(* CODESYS project testLD_RECOVERED_2018-03-27T13-50-33.project

Project tree, tasks and I/O mapping:
  Device : Jinan Cherry-ARM Cortex-VxWorks, Jinan Cheery Electric Co., Ltd., version 3.5.11.20
    application Application
      libraries: Standard, * (System)
      task MainTask (cyclic, interval 4 ms, priority 1) calls PLC_PRG
      task EtherCAT_Task (cyclic, interval t#4ms, priority 1) calls nothing
      program PLC_PRG [FBD]
    SoftMotion General Axis Pool
    EtherCAT_Master : EtherCAT Master, 3S - Smart Software Solutions GmbH, version 3.5.12.0
        settings: NetworkName = 'gem1'; NetworkName = "gem1"; SrcAddress1 = 10; SrcAddress2 = 889192739
      FR8200 : EtherCAT Adapter, Huatai-smartLink, order no. FR8200, version Revision=16#00010001
          settings: ModularDevice = True; Number of Outputs = 0; Number of Inputs = 0; Number of Infos about Outputs = 0; Number of Infos about Inputs = 0; MDP_InputOffsets = [0,0,32,64,80]; MDP_OutputOffsets = [0,0,0,0,16]; StationAlias = 0; Sync.Length = 4; Sync.Length = 12; FMMU.Length = 4; FMMU.Length = 12; Number of RxPDOs of the Slave = 2; Number of TxPDOs of the Slave = 4; DC sync0 cycletime = 4000; DC sync1 cycletime = 4000; Number of SDO = 4; Command_0.Index = 16#8000; Command_0.Subindex = 16#01; Command_0.Value = 6; Command_0.Size = 16; Command_0.AbortIfError = FALSE; Command_0.JumpToLine = FALSE; Command_0.Line = 0; Command_0.CompleteAccess = False; Command_0.Index = 16#8010; Command_0.Subindex = 16#01; Command_0.Value = 6; Command_0.Size = 16; Command_0.AbortIfError = FALSE; Command_0.JumpToLine = FALSE; Command_0.Line = 0; Command_0.CompleteAccess = False; Command_0.Index = 16#8020; Command_0.Subindex = 16#01; Command_0.Value = 12; Command_0.Size = 16; Command_0.AbortIfError = FALSE; Command_0.JumpToLine = FALSE; Command_0.Line = 0;
            Command_0.CompleteAccess = False; Command_0.Index = 16#8030; Command_0.Subindex = 16#01; Command_0.Value = 12; Command_0.Size = 16; Command_0.AbortIfError = FALSE; Command_0.JumpToLine = FALSE; Command_0.Line = 0; Command_0.CompleteAccess = False; RxTxPdo.NumberofExcludes = 0; RxTxPdo.NumberofEntries = 9; RxTxPdo.Index = 16#1602; RxTxPdo.Fixed = False; RxTxPdo.Mandatory = False; RxTxPdo.Virtual = False; RxTxPdo.Sm = 2; RxTxPdo.Su = 0; RxTxPdo.Name = 'Channels Data'; RxTxPdo.DependOnSlot = True; RxTxPdo.DependOnSlotGroup = False; RxTxPdo.OverwrittenByModule = True; Channel 1.Index = 16#7040; Channel 1.SubIndex = 1; Channel 1.Size = 1; Channel 1.Offset = 0; Channel 1.DependOnSlot = True; Channel 1.DependOnSlotGroup = True; Channel 2.Index = 16#7040; Channel 2.SubIndex = 2; Channel 2.Size = 1; Channel 2.Offset = 0; Channel 2.DependOnSlot = True; Channel 2.DependOnSlotGroup = True; Channel 3.Index = 16#7040; Channel 3.SubIndex = 3; Channel 3.Size = 1; Channel 3.Offset = 0; Channel 3.DependOnSlot = True; Channel 3.DependOnSlotGroup = True; Channel 4.Index = 16#7040;
            Channel 4.SubIndex = 4; Channel 4.Size = 1; Channel 4.Offset = 0; Channel 4.DependOnSlot = True; Channel 4.DependOnSlotGroup = True; Channel 5.Index = 16#7040; Channel 5.SubIndex = 5; Channel 5.Size = 1; Channel 5.Offset = 0; Channel 5.DependOnSlot = True; Channel 5.DependOnSlotGroup = True; Channel 6.Index = 16#7040; Channel 6.SubIndex = 6; Channel 6.Size = 1; Channel 6.Offset = 0; Channel 6.DependOnSlot = True; Channel 6.DependOnSlotGroup = True; Channel 7.Index = 16#7040; Channel 7.SubIndex = 7; Channel 7.Size = 1; Channel 7.Offset = 0; Channel 7.DependOnSlot = True; Channel 7.DependOnSlotGroup = True; Channel 8.Index = 16#7040; Channel 8.SubIndex = 8; Channel 8.Size = 1; Channel 8.Offset = 0; Channel 8.DependOnSlot = True; Channel 8.DependOnSlotGroup = True; Entry.Index = 16#0000; Entry.SubIndex = 9; Entry.Size = 8; Entry.Offset = 0; Entry.DependOnSlot = True; Entry.DependOnSlotGroup = True; RxTxPdo.NumberofExcludes = 0; RxTxPdo.NumberofEntries = 9; RxTxPdo.Index = 16#1603; RxTxPdo.Fixed = False; RxTxPdo.Mandatory = False;
            RxTxPdo.Virtual = False; RxTxPdo.Sm = 2; RxTxPdo.Su = 0; RxTxPdo.Name = 'Channels Data'; RxTxPdo.DependOnSlot = True; RxTxPdo.DependOnSlotGroup = False; RxTxPdo.OverwrittenByModule = True; Channel 1.Index = 16#7030; Channel 1.SubIndex = 1; Channel 1.Size = 1; Channel 1.Offset = 0; Channel 1.DependOnSlot = True; Channel 1.DependOnSlotGroup = True; Channel 2.Index = 16#7030; Channel 2.SubIndex = 2; Channel 2.Size = 1; Channel 2.Offset = 0; Channel 2.DependOnSlot = True; Channel 2.DependOnSlotGroup = True; Channel 3.Index = 16#7030; Channel 3.SubIndex = 3; Channel 3.Size = 1; Channel 3.Offset = 0; Channel 3.DependOnSlot = True; Channel 3.DependOnSlotGroup = True; Channel 4.Index = 16#7030; Channel 4.SubIndex = 4; Channel 4.Size = 1; Channel 4.Offset = 0; Channel 4.DependOnSlot = True; Channel 4.DependOnSlotGroup = True; Channel 5.Index = 16#7030; Channel 5.SubIndex = 5; Channel 5.Size = 1; Channel 5.Offset = 0; Channel 5.DependOnSlot = True; Channel 5.DependOnSlotGroup = True; Channel 6.Index = 16#7030; Channel 6.SubIndex = 6; Channel 6.Size = 1;
            Channel 6.Offset = 0; Channel 6.DependOnSlot = True; Channel 6.DependOnSlotGroup = True; Channel 7.Index = 16#7030; Channel 7.SubIndex = 7; Channel 7.Size = 1; Channel 7.Offset = 0; Channel 7.DependOnSlot = True; Channel 7.DependOnSlotGroup = True; Channel 8.Index = 16#7030; Channel 8.SubIndex = 8; Channel 8.Size = 1; Channel 8.Offset = 0; Channel 8.DependOnSlot = True; Channel 8.DependOnSlotGroup = True; Entry.Index = 16#0000; Entry.SubIndex = 9; Entry.Size = 8; Entry.Offset = 0; Entry.DependOnSlot = True; Entry.DependOnSlotGroup = True; RxTxPdo.NumberofExcludes = 0; RxTxPdo.NumberofEntries = 12; RxTxPdo.Index = 16#1A00; RxTxPdo.Fixed = False; RxTxPdo.Mandatory = False; RxTxPdo.Virtual = False; RxTxPdo.Sm = 3; RxTxPdo.Su = 0; RxTxPdo.Name = 'Channels Data'; RxTxPdo.DependOnSlot = True; RxTxPdo.DependOnSlotGroup = False; RxTxPdo.OverwrittenByModule = True; Channel 1.Index = 16#6000; Channel 1.SubIndex = 1; Channel 1.Size = 1; Channel 1.Offset = 0; Channel 1.DependOnSlot = True; Channel 1.DependOnSlotGroup = True; Channel 2.Index = 16#6000;
            Channel 2.SubIndex = 2; Channel 2.Size = 1; Channel 2.Offset = 0; Channel 2.DependOnSlot = True; Channel 2.DependOnSlotGroup = True; Channel 3.Index = 16#6000; Channel 3.SubIndex = 3; Channel 3.Size = 1; Channel 3.Offset = 0; Channel 3.DependOnSlot = True; Channel 3.DependOnSlotGroup = True; Channel 4.Index = 16#6000; Channel 4.SubIndex = 4; Channel 4.Size = 1; Channel 4.Offset = 0; Channel 4.DependOnSlot = True; Channel 4.DependOnSlotGroup = True; Channel 5.Index = 16#6000; Channel 5.SubIndex = 5; Channel 5.Size = 1; Channel 5.Offset = 0; Channel 5.DependOnSlot = True; Channel 5.DependOnSlotGroup = True; Channel 6.Index = 16#6000; Channel 6.SubIndex = 6; Channel 6.Size = 1; Channel 6.Offset = 0; Channel 6.DependOnSlot = True; Channel 6.DependOnSlotGroup = True; Channel 7.Index = 16#6000; Channel 7.SubIndex = 7; Channel 7.Size = 1; Channel 7.Offset = 0; Channel 7.DependOnSlot = True; Channel 7.DependOnSlotGroup = True; Channel 8.Index = 16#6000; Channel 8.SubIndex = 8; Channel 8.Size = 1; Channel 8.Offset = 0; Channel 8.DependOnSlot = True;
            Channel 8.DependOnSlotGroup = True; Entry.Index = 16#0000; Entry.SubIndex = 9; Entry.Size = 8; Entry.Offset = 0; Entry.DependOnSlot = True; Entry.DependOnSlotGroup = True; Temperature Alarm.Index = 16#6002; Temperature Alarm.SubIndex = 1; Temperature Alarm.Size = 1; Temperature Alarm.Offset = 0; Temperature Alarm.DependOnSlot = True; Temperature Alarm.DependOnSlotGroup = True; Voltage Alarm.Index = 16#6002; Voltage Alarm.SubIndex = 2; Voltage Alarm.Size = 1; Voltage Alarm.Offset = 0; Voltage Alarm.DependOnSlot = True; Voltage Alarm.DependOnSlotGroup = True; Entry.Index = 16#0000; Entry.SubIndex = 3; Entry.Size = 14; Entry.Offset = 0; Entry.DependOnSlot = False; Entry.DependOnSlotGroup = False; RxTxPdo.NumberofExcludes = 0; RxTxPdo.NumberofEntries = 12; RxTxPdo.Index = 16#1A01; RxTxPdo.Fixed = False; RxTxPdo.Mandatory = False; RxTxPdo.Virtual = False; RxTxPdo.Sm = 3; RxTxPdo.Su = 0; RxTxPdo.Name = 'Channels Data'; RxTxPdo.DependOnSlot = True; RxTxPdo.DependOnSlotGroup = False; RxTxPdo.OverwrittenByModule = True; Channel 1.Index = 16#6010; Channel 1.SubIndex = 1; Channel 1.Size = 1;
            Channel 1.Offset = 0; Channel 1.DependOnSlot = True; Channel 1.DependOnSlotGroup = True; Channel 2.Index = 16#6010; Channel 2.SubIndex = 2; Channel 2.Size = 1; Channel 2.Offset = 0; Channel 2.DependOnSlot = True; Channel 2.DependOnSlotGroup = True; Channel 3.Index = 16#6010; Channel 3.SubIndex = 3; Channel 3.Size = 1; Channel 3.Offset = 0; Channel 3.DependOnSlot = True; Channel 3.DependOnSlotGroup = True; Channel 4.Index = 16#6010; Channel 4.SubIndex = 4; Channel 4.Size = 1; Channel 4.Offset = 0; Channel 4.DependOnSlot = True; Channel 4.DependOnSlotGroup = True; Channel 5.Index = 16#6010; Channel 5.SubIndex = 5; Channel 5.Size = 1; Channel 5.Offset = 0; Channel 5.DependOnSlot = True; Channel 5.DependOnSlotGroup = True; Channel 6.Index = 16#6010; Channel 6.SubIndex = 6; Channel 6.Size = 1; Channel 6.Offset = 0; Channel 6.DependOnSlot = True; Channel 6.DependOnSlotGroup = True; Channel 7.Index = 16#6010; Channel 7.SubIndex = 7; Channel 7.Size = 1; Channel 7.Offset = 0; Channel 7.DependOnSlot = True; Channel 7.DependOnSlotGroup = True; Channel 8.Index = 16#6010;
            Channel 8.SubIndex = 8; Channel 8.Size = 1; Channel 8.Offset = 0; Channel 8.DependOnSlot = True; Channel 8.DependOnSlotGroup = True; Entry.Index = 16#0000; Entry.SubIndex = 9; Entry.Size = 8; Entry.Offset = 0; Entry.DependOnSlot = True; Entry.DependOnSlotGroup = True; Temperature Alarm.Index = 16#6012; Temperature Alarm.SubIndex = 1; Temperature Alarm.Size = 1; Temperature Alarm.Offset = 0; Temperature Alarm.DependOnSlot = True; Temperature Alarm.DependOnSlotGroup = True; Voltage Alarm.Index = 16#6012; Voltage Alarm.SubIndex = 2; Voltage Alarm.Size = 1; Voltage Alarm.Offset = 0; Voltage Alarm.DependOnSlot = True; Voltage Alarm.DependOnSlotGroup = True; Entry.Index = 16#0000; Entry.SubIndex = 3; Entry.Size = 14; Entry.Offset = 0; Entry.DependOnSlot = False; Entry.DependOnSlotGroup = False; RxTxPdo.NumberofExcludes = 0; RxTxPdo.NumberofEntries = 3; RxTxPdo.Index = 16#1A02; RxTxPdo.Fixed = False; RxTxPdo.Mandatory = False; RxTxPdo.Virtual = False; RxTxPdo.Sm = 3; RxTxPdo.Su = 0; RxTxPdo.Name = 'Alarm Data'; RxTxPdo.DependOnSlot = True; RxTxPdo.DependOnSlotGroup = False;
            RxTxPdo.OverwrittenByModule = True; Temperature Alarm.Index = 16#6022; Temperature Alarm.SubIndex = 1; Temperature Alarm.Size = 1; Temperature Alarm.Offset = 0; Temperature Alarm.DependOnSlot = True; Temperature Alarm.DependOnSlotGroup = True; Voltage Alarm.Index = 16#6022; Voltage Alarm.SubIndex = 2; Voltage Alarm.Size = 1; Voltage Alarm.Offset = 0; Voltage Alarm.DependOnSlot = True; Voltage Alarm.DependOnSlotGroup = True; Entry.Index = 16#0000; Entry.SubIndex = 3; Entry.Size = 14; Entry.Offset = 0; Entry.DependOnSlot = False; Entry.DependOnSlotGroup = False; RxTxPdo.NumberofExcludes = 0; RxTxPdo.NumberofEntries = 3; RxTxPdo.Index = 16#1A03; RxTxPdo.Fixed = False; RxTxPdo.Mandatory = False; RxTxPdo.Virtual = False; RxTxPdo.Sm = 3; RxTxPdo.Su = 0; RxTxPdo.Name = 'Alarm Data'; RxTxPdo.DependOnSlot = True; RxTxPdo.DependOnSlotGroup = False; RxTxPdo.OverwrittenByModule = True; Temperature Alarm.Index = 16#6032; Temperature Alarm.SubIndex = 1; Temperature Alarm.Size = 1; Temperature Alarm.Offset = 0; Temperature Alarm.DependOnSlot = True; Temperature Alarm.DependOnSlotGroup = True; Voltage Alarm.Index = 16#6032; Voltage Alarm.SubIndex = 2; Voltage Alarm.Size = 1;
            Voltage Alarm.Offset = 0; Voltage Alarm.DependOnSlot = True; Voltage Alarm.DependOnSlotGroup = True; Entry.Index = 16#0000; Entry.SubIndex = 3; Entry.Size = 14; Entry.Offset = 0; Entry.DependOnSlot = False; Entry.DependOnSlotGroup = False; Channel 1.Name = 'Channel 1'; Channel 1.DataType = 'BOOL'; Channel 1.Default = ''; Channel 1.Comment = ''; Channel 2.Name = 'Channel 2'; Channel 2.DataType = 'BOOL'; Channel 2.Default = ''; Channel 2.Comment = ''; Channel 3.Name = 'Channel 3'; Channel 3.DataType = 'BOOL'; Channel 3.Default = ''; Channel 3.Comment = ''; Channel 4.Name = 'Channel 4'; Channel 4.DataType = 'BOOL'; Channel 4.Default = ''; Channel 4.Comment = ''; Channel 5.Name = 'Channel 5'; Channel 5.DataType = 'BOOL'; Channel 5.Default = ''; Channel 5.Comment = ''; Channel 6.Name = 'Channel 6'; Channel 6.DataType = 'BOOL'; Channel 6.Default = ''; Channel 6.Comment = ''; Channel 7.Name = 'Channel 7'; Channel 7.DataType = 'BOOL'; Channel 7.Default = ''; Channel 7.Comment = ''; Channel 8.Name = 'Channel 8'; Channel 8.DataType = 'BOOL'; Channel 8.Default = '';
            Channel 8.Comment = ''; Entry.Name = ''; Entry.DataType = ''; Entry.Default = ''; Entry.Comment = ''; Channel 1.Name = 'Channel 1'; Channel 1.DataType = 'BOOL'; Channel 1.Default = ''; Channel 1.Comment = ''; Channel 2.Name = 'Channel 2'; Channel 2.DataType = 'BOOL'; Channel 2.Default = ''; Channel 2.Comment = ''; Channel 3.Name = 'Channel 3'; Channel 3.DataType = 'BOOL'; Channel 3.Default = ''; Channel 3.Comment = ''; Channel 4.Name = 'Channel 4'; Channel 4.DataType = 'BOOL'; Channel 4.Default = ''; Channel 4.Comment = ''; Channel 5.Name = 'Channel 5'; Channel 5.DataType = 'BOOL'; Channel 5.Default = ''; Channel 5.Comment = ''; Channel 6.Name = 'Channel 6'; Channel 6.DataType = 'BOOL'; Channel 6.Default = ''; Channel 6.Comment = ''; Channel 7.Name = 'Channel 7'; Channel 7.DataType = 'BOOL'; Channel 7.Default = ''; Channel 7.Comment = ''; Channel 8.Name = 'Channel 8'; Channel 8.DataType = 'BOOL'; Channel 8.Default = ''; Channel 8.Comment = ''; Entry.Name = ''; Entry.DataType = ''; Entry.Default = '';
            Entry.Comment = ''; Channel 1.Name = 'Channel 1'; Channel 1.DataType = 'BOOL'; Channel 1.Default = ''; Channel 1.Comment = ''; Channel 2.Name = 'Channel 2'; Channel 2.DataType = 'BOOL'; Channel 2.Default = ''; Channel 2.Comment = ''; Channel 3.Name = 'Channel 3'; Channel 3.DataType = 'BOOL'; Channel 3.Default = ''; Channel 3.Comment = ''; Channel 4.Name = 'Channel 4'; Channel 4.DataType = 'BOOL'; Channel 4.Default = ''; Channel 4.Comment = ''; Channel 5.Name = 'Channel 5'; Channel 5.DataType = 'BOOL'; Channel 5.Default = ''; Channel 5.Comment = ''; Channel 6.Name = 'Channel 6'; Channel 6.DataType = 'BOOL'; Channel 6.Default = ''; Channel 6.Comment = ''; Channel 7.Name = 'Channel 7'; Channel 7.DataType = 'BOOL'; Channel 7.Default = ''; Channel 7.Comment = ''; Channel 8.Name = 'Channel 8'; Channel 8.DataType = 'BOOL'; Channel 8.Default = ''; Channel 8.Comment = ''; Entry.Name = ''; Entry.DataType = ''; Entry.Default = ''; Entry.Comment = ''; Temperature Alarm.Name = 'Temperature Alarm'; Temperature Alarm.DataType = 'BOOL'; Temperature Alarm.Default = '';
            Temperature Alarm.Comment = ''; Voltage Alarm.Name = 'Voltage Alarm'; Voltage Alarm.DataType = 'BOOL'; Voltage Alarm.Default = ''; Voltage Alarm.Comment = ''; Entry.Name = ''; Entry.DataType = ''; Entry.Default = ''; Entry.Comment = ''; Channel 1.Name = 'Channel 1'; Channel 1.DataType = 'BOOL'; Channel 1.Default = ''; Channel 1.Comment = ''; Channel 2.Name = 'Channel 2'; Channel 2.DataType = 'BOOL'; Channel 2.Default = ''; Channel 2.Comment = ''; Channel 3.Name = 'Channel 3'; Channel 3.DataType = 'BOOL'; Channel 3.Default = ''; Channel 3.Comment = ''; Channel 4.Name = 'Channel 4'; Channel 4.DataType = 'BOOL'; Channel 4.Default = ''; Channel 4.Comment = ''; Channel 5.Name = 'Channel 5'; Channel 5.DataType = 'BOOL'; Channel 5.Default = ''; Channel 5.Comment = ''; Channel 6.Name = 'Channel 6'; Channel 6.DataType = 'BOOL'; Channel 6.Default = ''; Channel 6.Comment = ''; Channel 7.Name = 'Channel 7'; Channel 7.DataType = 'BOOL'; Channel 7.Default = ''; Channel 7.Comment = ''; Channel 8.Name = 'Channel 8'; Channel 8.DataType = 'BOOL'; Channel 8.Default = '';
            Channel 8.Comment = ''; Entry.Name = ''; Entry.DataType = ''; Entry.Default = ''; Entry.Comment = ''; Temperature Alarm.Name = 'Temperature Alarm'; Temperature Alarm.DataType = 'BOOL'; Temperature Alarm.Default = ''; Temperature Alarm.Comment = ''; Voltage Alarm.Name = 'Voltage Alarm'; Voltage Alarm.DataType = 'BOOL'; Voltage Alarm.Default = ''; Voltage Alarm.Comment = ''; Entry.Name = ''; Entry.DataType = ''; Entry.Default = ''; Entry.Comment = ''; Temperature Alarm.Name = 'Temperature Alarm'; Temperature Alarm.DataType = 'BOOL'; Temperature Alarm.Default = ''; Temperature Alarm.Comment = ''; Voltage Alarm.Name = 'Voltage Alarm'; Voltage Alarm.DataType = 'BOOL'; Voltage Alarm.Default = ''; Voltage Alarm.Comment = ''; Entry.Name = ''; Entry.DataType = ''; Entry.Default = ''; Entry.Comment = ''; Temperature Alarm.Name = 'Temperature Alarm'; Temperature Alarm.DataType = 'BOOL'; Temperature Alarm.Default = ''; Temperature Alarm.Comment = ''; Voltage Alarm.Name = 'Voltage Alarm'; Voltage Alarm.DataType = 'BOOL'; Voltage Alarm.Default = ''; Voltage Alarm.Comment = ''; Entry.Name = ''; Entry.DataType = ''; Entry.Default = '';
            Entry.Comment = ''
        <空14>
        <空10>
        <空19>
        <空32>
        <空23>
        <空15>
        <空21>
        <空31>
        <空26>
        <空16>
        <空20>
        FR1118 : FR Serials IO Modules, Huatai-smartLink, order no. FR1118, version 0
            settings: Number of Inputs = 25; Number of Infos about Inputs = 25; Channel 1.Offset = 0; Channel 1.DependOnSlot = True; Channel 1.DependOnSlotGroup = True; Channel 2.Offset = 0; Channel 2.DependOnSlot = True; Channel 2.DependOnSlotGroup = True; Channel 3.Offset = 0; Channel 3.DependOnSlot = True; Channel 3.DependOnSlotGroup = True; Channel 4.Offset = 0; Channel 4.DependOnSlot = True; Channel 4.DependOnSlotGroup = True; Channel 5.Offset = 0; Channel 5.DependOnSlot = True; Channel 5.DependOnSlotGroup = True; Channel 6.Offset = 0; Channel 6.DependOnSlot = True; Channel 6.DependOnSlotGroup = True; Channel 7.Offset = 0; Channel 7.DependOnSlot = True; Channel 7.DependOnSlotGroup = True; Channel 8.Offset = 0; Channel 8.DependOnSlot = True; Channel 8.DependOnSlotGroup = True; Entry.Offset = 0; Entry.DependOnSlot = True; Entry.DependOnSlotGroup = True; Temperature Alarm.Offset = 0; Temperature Alarm.DependOnSlot = True; Temperature Alarm.DependOnSlotGroup = True; Voltage Alarm.Offset = 0; Voltage Alarm.DependOnSlot = True; Voltage Alarm.DependOnSlotGroup = True; Entry.Offset = 0; Entry.DependOnSlot = False; Entry.DependOnSlotGroup = False; Channel 1.Default = ''; Channel 2.Default = '';
              Channel 3.Default = ''; Channel 4.Default = ''; Channel 5.Default = ''; Channel 6.Default = ''; Channel 7.Default = ''; Channel 8.Default = ''; Entry.Name = ''; Entry.DataType = ''; Entry.Default = ''; Temperature Alarm.Default = ''; Voltage Alarm.Default = ''; Entry.Name = ''; Entry.DataType = ''; Entry.Default = ''
            unmapped channels: Channel 1, Channel 2, Channel 3, Channel 4, Channel 5, Channel 6, Channel 7, Channel 8, , Temperature Alarm, Voltage Alarm, , , , , , , , , , , , , , 
        <空29>
        FR1118_1 : FR Serials IO Modules, Huatai-smartLink, order no. FR1118, version 0
            settings: Number of Inputs = 25; Number of Infos about Inputs = 25; Channel 1.Index = 16#6010; Channel 1.SubIndex = 1; Channel 1.Size = 1; Channel 1.Offset = 0; Channel 1.DependOnSlot = True; Channel 1.DependOnSlotGroup = True; Channel 2.Index = 16#6010; Channel 2.SubIndex = 2; Channel 2.Size = 1; Channel 2.Offset = 0; Channel 2.DependOnSlot = True; Channel 2.DependOnSlotGroup = True; Channel 3.Index = 16#6010; Channel 3.SubIndex = 3; Channel 3.Size = 1; Channel 3.Offset = 0; Channel 3.DependOnSlot = True; Channel 3.DependOnSlotGroup = True; Channel 4.Index = 16#6010; Channel 4.SubIndex = 4; Channel 4.Size = 1; Channel 4.Offset = 0; Channel 4.DependOnSlot = True; Channel 4.DependOnSlotGroup = True; Channel 5.Index = 16#6010; Channel 5.SubIndex = 5; Channel 5.Size = 1; Channel 5.Offset = 0; Channel 5.DependOnSlot = True; Channel 5.DependOnSlotGroup = True; Channel 6.Index = 16#6010; Channel 6.SubIndex = 6; Channel 6.Size = 1; Channel 6.Offset = 0; Channel 6.DependOnSlot = True; Channel 6.DependOnSlotGroup = True; Channel 7.Index = 16#6010; Channel 7.SubIndex = 7;
              Channel 7.Size = 1; Channel 7.Offset = 0; Channel 7.DependOnSlot = True; Channel 7.DependOnSlotGroup = True; Channel 8.Index = 16#6010; Channel 8.SubIndex = 8; Channel 8.Size = 1; Channel 8.Offset = 0; Channel 8.DependOnSlot = True; Channel 8.DependOnSlotGroup = True; Entry.Index = 16#0000; Entry.SubIndex = 9; Entry.Size = 8; Entry.Offset = 0; Entry.DependOnSlot = True; Entry.DependOnSlotGroup = True; Temperature Alarm.Index = 16#6012; Temperature Alarm.SubIndex = 1; Temperature Alarm.Size = 1; Temperature Alarm.Offset = 0; Temperature Alarm.DependOnSlot = True; Temperature Alarm.DependOnSlotGroup = True; Voltage Alarm.Index = 16#6012; Voltage Alarm.SubIndex = 2; Voltage Alarm.Size = 1; Voltage Alarm.Offset = 0; Voltage Alarm.DependOnSlot = True; Voltage Alarm.DependOnSlotGroup = True; Entry.Index = 16#0000; Entry.SubIndex = 3; Entry.Size = 14; Entry.Offset = 0; Entry.DependOnSlot = False; Entry.DependOnSlotGroup = False; Channel 1.Name = 'Channel 1'; Channel 1.DataType = 'BOOL'; Channel 1.Default = ''; Channel 1.Comment = ''; Channel 2.Name = 'Channel 2'; Channel 2.DataType = 'BOOL';
              Channel 2.Default = ''; Channel 2.Comment = ''; Channel 3.Name = 'Channel 3'; Channel 3.DataType = 'BOOL'; Channel 3.Default = ''; Channel 3.Comment = ''; Channel 4.Name = 'Channel 4'; Channel 4.DataType = 'BOOL'; Channel 4.Default = ''; Channel 4.Comment = ''; Channel 5.Name = 'Channel 5'; Channel 5.DataType = 'BOOL'; Channel 5.Default = ''; Channel 5.Comment = ''; Channel 6.Name = 'Channel 6'; Channel 6.DataType = 'BOOL'; Channel 6.Default = ''; Channel 6.Comment = ''; Channel 7.Name = 'Channel 7'; Channel 7.DataType = 'BOOL'; Channel 7.Default = ''; Channel 7.Comment = ''; Channel 8.Name = 'Channel 8'; Channel 8.DataType = 'BOOL'; Channel 8.Default = ''; Channel 8.Comment = ''; Entry.Name = ''; Entry.DataType = ''; Entry.Default = ''; Entry.Comment = ''; Temperature Alarm.Name = 'Temperature Alarm'; Temperature Alarm.DataType = 'BOOL'; Temperature Alarm.Default = ''; Temperature Alarm.Comment = ''; Voltage Alarm.Name = 'Voltage Alarm'; Voltage Alarm.DataType = 'BOOL'; Voltage Alarm.Default = ''; Voltage Alarm.Comment = ''; Entry.Name = ''; Entry.DataType = '';
              Entry.Default = ''; Entry.Comment = ''
            unmapped channels: Channel 1, Channel 2, Channel 3, Channel 4, Channel 5, Channel 6, Channel 7, Channel 8, , Temperature Alarm, Voltage Alarm, , , , , , , , , , , , , , 
        <空18>
        <空22>
        <空7>
        <空5>
        <空11>
        FR2118_1 : FR Serials IO Modules, Huatai-smartLink, order no. FR2118, version 0
            settings: Number of Outputs = 9; Number of Inputs = 16; Number of Infos about Outputs = 9; Number of Infos about Inputs = 16; Channel 1.Index = 16#7030; Channel 1.SubIndex = 1; Channel 1.Size = 1; Channel 1.Offset = 0; Channel 1.DependOnSlot = True; Channel 1.DependOnSlotGroup = True; Channel 2.Index = 16#7030; Channel 2.SubIndex = 2; Channel 2.Size = 1; Channel 2.Offset = 0; Channel 2.DependOnSlot = True; Channel 2.DependOnSlotGroup = True; Channel 3.Index = 16#7030; Channel 3.SubIndex = 3; Channel 3.Size = 1; Channel 3.Offset = 0; Channel 3.DependOnSlot = True; Channel 3.DependOnSlotGroup = True; Channel 4.Index = 16#7030; Channel 4.SubIndex = 4; Channel 4.Size = 1; Channel 4.Offset = 0; Channel 4.DependOnSlot = True; Channel 4.DependOnSlotGroup = True; Channel 5.Index = 16#7030; Channel 5.SubIndex = 5; Channel 5.Size = 1; Channel 5.Offset = 0; Channel 5.DependOnSlot = True; Channel 5.DependOnSlotGroup = True; Channel 6.Index = 16#7030; Channel 6.SubIndex = 6; Channel 6.Size = 1; Channel 6.Offset = 0; Channel 6.DependOnSlot = True; Channel 6.DependOnSlotGroup = True;
              Channel 7.Index = 16#7030; Channel 7.SubIndex = 7; Channel 7.Size = 1; Channel 7.Offset = 0; Channel 7.DependOnSlot = True; Channel 7.DependOnSlotGroup = True; Channel 8.Index = 16#7030; Channel 8.SubIndex = 8; Channel 8.Size = 1; Channel 8.Offset = 0; Channel 8.DependOnSlot = True; Channel 8.DependOnSlotGroup = True; Entry.Index = 16#0000; Entry.SubIndex = 9; Entry.Size = 8; Entry.Offset = 0; Entry.DependOnSlot = True; Entry.DependOnSlotGroup = True; Temperature Alarm.Index = 16#6032; Temperature Alarm.SubIndex = 1; Temperature Alarm.Size = 1; Temperature Alarm.Offset = 0; Temperature Alarm.DependOnSlot = True; Temperature Alarm.DependOnSlotGroup = True; Voltage Alarm.Index = 16#6032; Voltage Alarm.SubIndex = 2; Voltage Alarm.Size = 1; Voltage Alarm.Offset = 0; Voltage Alarm.DependOnSlot = True; Voltage Alarm.DependOnSlotGroup = True; Entry.Index = 16#0000; Entry.SubIndex = 3; Entry.Size = 14; Entry.Offset = 0; Entry.DependOnSlot = False; Entry.DependOnSlotGroup = False; Channel 1.Name = 'Channel 1'; Channel 1.DataType = 'BOOL'; Channel 1.Default = ''; Channel 1.Comment = '';
              Channel 2.Name = 'Channel 2'; Channel 2.DataType = 'BOOL'; Channel 2.Default = ''; Channel 2.Comment = ''; Channel 3.Name = 'Channel 3'; Channel 3.DataType = 'BOOL'; Channel 3.Default = ''; Channel 3.Comment = ''; Channel 4.Name = 'Channel 4'; Channel 4.DataType = 'BOOL'; Channel 4.Default = ''; Channel 4.Comment = ''; Channel 5.Name = 'Channel 5'; Channel 5.DataType = 'BOOL'; Channel 5.Default = ''; Channel 5.Comment = ''; Channel 6.Name = 'Channel 6'; Channel 6.DataType = 'BOOL'; Channel 6.Default = ''; Channel 6.Comment = ''; Channel 7.Name = 'Channel 7'; Channel 7.DataType = 'BOOL'; Channel 7.Default = ''; Channel 7.Comment = ''; Channel 8.Name = 'Channel 8'; Channel 8.DataType = 'BOOL'; Channel 8.Default = ''; Channel 8.Comment = ''; Entry.Name = ''; Entry.DataType = ''; Entry.Default = ''; Entry.Comment = ''; Temperature Alarm.Name = 'Temperature Alarm'; Temperature Alarm.DataType = 'BOOL'; Temperature Alarm.Default = ''; Temperature Alarm.Comment = ''; Voltage Alarm.Name = 'Voltage Alarm'; Voltage Alarm.DataType = 'BOOL'; Voltage Alarm.Default = ''; Voltage Alarm.Comment = '';
              Entry.Name = ''; Entry.DataType = ''; Entry.Default = ''; Entry.Comment = ''
            output Application.PLC_PRG.Out1 : BIT  // Channel 1
            unmapped channels: Channel 2, Channel 3, Channel 4, Channel 5, Channel 6, Channel 7, Channel 8, , Temperature Alarm, Voltage Alarm, , , , , , , , , , , , , , 
        <空24>
        FR2118 : FR Serials IO Modules, Huatai-smartLink, order no. FR2118, version 0
            settings: Number of Outputs = 9; Number of Inputs = 16; Number of Infos about Outputs = 9; Number of Infos about Inputs = 16; Channel 1.Index = 16#7020; Channel 1.Offset = 0; Channel 1.DependOnSlot = True; Channel 1.DependOnSlotGroup = True; Channel 2.Index = 16#7020; Channel 2.Offset = 0; Channel 2.DependOnSlot = True; Channel 2.DependOnSlotGroup = True; Channel 3.Index = 16#7020; Channel 3.Offset = 0; Channel 3.DependOnSlot = True; Channel 3.DependOnSlotGroup = True; Channel 4.Index = 16#7020; Channel 4.Offset = 0; Channel 4.DependOnSlot = True; Channel 4.DependOnSlotGroup = True; Channel 5.Index = 16#7020; Channel 5.Offset = 0; Channel 5.DependOnSlot = True; Channel 5.DependOnSlotGroup = True; Channel 6.Index = 16#7020; Channel 6.Offset = 0; Channel 6.DependOnSlot = True; Channel 6.DependOnSlotGroup = True; Channel 7.Index = 16#7020; Channel 7.Offset = 0; Channel 7.DependOnSlot = True; Channel 7.DependOnSlotGroup = True; Channel 8.Index = 16#7020; Channel 8.Offset = 0; Channel 8.DependOnSlot = True; Channel 8.DependOnSlotGroup = True; Entry.Offset = 0; Entry.DependOnSlot = True; Entry.DependOnSlotGroup = True; Temperature Alarm.Index = 16#6022;
              Temperature Alarm.SubIndex = 1; Temperature Alarm.Size = 1; Temperature Alarm.Offset = 0; Temperature Alarm.DependOnSlot = True; Temperature Alarm.DependOnSlotGroup = True; Voltage Alarm.Index = 16#6022; Voltage Alarm.SubIndex = 2; Voltage Alarm.Size = 1; Voltage Alarm.Offset = 0; Voltage Alarm.DependOnSlot = True; Voltage Alarm.DependOnSlotGroup = True; Entry.Index = 16#0000; Entry.SubIndex = 3; Entry.Size = 14; Entry.Offset = 0; Entry.DependOnSlot = False; Entry.DependOnSlotGroup = False; Channel 1.Default = ''; Channel 2.Default = ''; Channel 3.Default = ''; Channel 4.Default = ''; Channel 5.Default = ''; Channel 6.Default = ''; Channel 7.Default = ''; Channel 8.Default = ''; Entry.Name = ''; Entry.DataType = ''; Entry.Default = ''; Temperature Alarm.Name = 'Temperature Alarm'; Temperature Alarm.DataType = 'BOOL'; Temperature Alarm.Default = ''; Temperature Alarm.Comment = ''; Voltage Alarm.Name = 'Voltage Alarm'; Voltage Alarm.DataType = 'BOOL'; Voltage Alarm.Default = ''; Voltage Alarm.Comment = ''; Entry.Name = ''; Entry.DataType = ''; Entry.Default = ''; Entry.Comment = ''
            output Application.PLC_PRG.Out1 : BIT  // Channel 1
            unmapped channels: Channel 2, Channel 3, Channel 4, Channel 5, Channel 6, Channel 7, Channel 8, , Temperature Alarm, Voltage Alarm, , , , , , , , , , , , , , 
        <空8>
        <空30>
        <空12>
        <空6>
        <空25>
        <空9>
        <空27>
        <空13>
        <空28>
        <空17>
*)

// Device/Application/PLC_PRG
PROGRAM PLC_PRG
VAR
	Out1: BOOL := false;
END_VAR

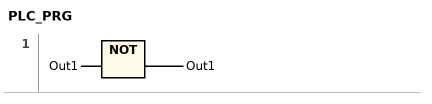
// NETWORK 1
Out1 := NOT Out1;

END_PROGRAM
